INTERFACE I_Observer

METHOD send_signal : BOOL
VAR_INPUT
	pAlarm		: POINTER TO FB_Alarm;
END_VAR
END_METHOD

END_INTERFACE

(* stored: Version 1.1.0.1, ProductVersion 3.1.4024.12
   Itf I_Observer: Id {4f3cef88-0c03-433a-a68e-c25d8f9a39f1}
   Method send_signal: Id {3d4aab7e-3102-477b-bc85-53b61297b67a} *)
